{attribute 'qualified_only'}
VAR_GLOBAL CONSTANT
    MaxCsvFields : INT := 99;
END_VAR

(* stored: Version 1.1.0.1, ProductVersion 3.1.4024.3
   GVL Param: Id {d0f6f374-0f52-07ff-3ed2-357cb320af4d}, ParameterList True *)
